TYPE ETherCAT_StatMonitor_VAR :
STRUCT
	//variables to be monitored // EthererCAT out  (IN for CLC)
	
	StatControlCMD : BessStateControl;
	OpModeControlCMD : BessOpmodeControl;
	//P Q references. 
	ActivePowerReference : DINT;
	ReactivePowerReference: DINT;
	Heartbeat : DINT;
	ClrAlarm : DINT;
	ClrFault : DINT;
	reserve1 : DINT;
	reserver2 : DINT;
	

		
END_STRUCT
END_TYPE

(* stored: Version 1.1.0.1, ProductVersion 3.1.4024.11
   DUT ETherCAT_StatMonitor_VAR: Id {213e5dbc-ec25-46dc-a36d-58b21fa6da93} *)
